TYPE U_NCI_STATE :
UNION

  stState             : ARRAY[1..MAX_NCI_CH] OF ST_NCI_STATE;

  byState   AT %i*    : ARRAY[1..MAX_NCI_CH] OF
                        ARRAY[1..SIZEOF(ST_NCI_STATE)] OF BYTE;
END_UNION
END_TYPE

(* stored: Version 1.1.0.1
   DUT U_NCI_STATE: Id {cfe88312-660b-41f8-a3a4-a04f87f8a037} *)
